FUNCTION_BLOCK AI_filter
VAR_INPUT
	AI 				:INT;
	MVF				:INT;
	Filtertid 		:INT;
	
END_VAR
VAR_OUTPUT
	MV				:INT;
END_VAR
VAR
	Filter1			: FB_BA_FltrPT1;
END_VAR
VAR // added by the converter: edge detectors and wires of the graphical bodies
    _w1, _w2 : ANY;
END_VAR


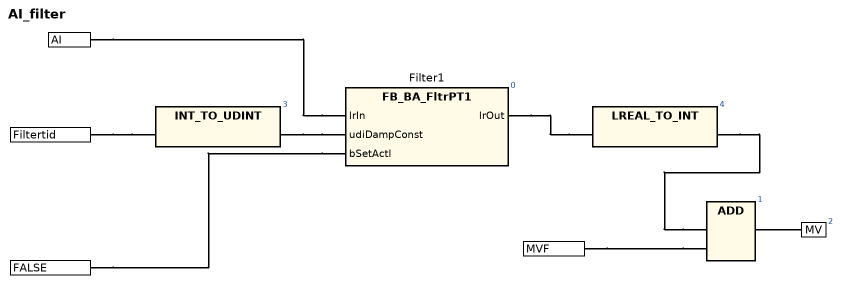
// PAGE
Filter1(lrIn := AI, udiDampConst := _w1, bSetActl := FALSE); // FB_BA_FltrPT1
MV := _w2 + MVF;
_w1 := INT_TO_UDINT(Filtertid);
_w2 := LREAL_TO_INT(Filter1.lrOut);

END_FUNCTION_BLOCK

(* stored: Version 1.1.0.1, ProductVersion 3.1.4020.12
   POU AI_filter: Id {5724d7e8-240c-4ca0-8a4e-b12fc82ec9f6}, SpecialFunc None *)
